FUNCTION TryConvert_SINT_TO_UINT : BOOL
VAR_INPUT
	in : SINT;
	out : REFERENCE TO UINT;
END_VAR

IF in < DatatypeLimits.MIN_VALUE_OF_SINT_WHICH_CAN_BE_HELD_IN_A_UINT THEN
	RETURN;
END_IF

out := SINT_TO_UINT(in);
TryConvert_SINT_TO_UINT := TRUE;

END_FUNCTION

(* stored: Version 1.1.0.1, ProductVersion 3.1.4024.12
   POU TryConvert_SINT_TO_UINT: Id {21f9fdf3-3100-4db6-ac32-0678241973a9}, SpecialFunc None *)
